PROGRAM MAIN
VAR
	// Invoker
	fbHMI_panel				: FB_ShowControlPanel;
	fbPendant_panel			: FB_ShowControlPanel;
	
	// Receiver
	fbFlyingHoist			: FB_FlyingHoist;
	refFlyingHoist			: REFERENCE TO FB_FlyingHoist := fbFlyingHoist;	
	fbFlameCannon			: FB_FlameCannon;
	refFlameCannon			: REFERENCE TO FB_FlameCannon := fbFlameCannon;	
	fbMovingHead			: FB_MovingHead;
	refMovingHead			: REFERENCE TO FB_MovingHead := fbMovingHead;	

	// Commands
	fbActorDownCommand			: FB_ActorDownCommand(refFlyingHoist);
	fbActorUpCommand			: FB_ActorUpCommand(refFlyingHoist);
	fbActorRotateCCWCommand		: FB_ActorRotateCCWCommand(refFlyingHoist);
	fbActorRotateCWCommand		: FB_ActorRotateCWCommand(refFlyingHoist);
	fbActorStopRotateCommand	: FB_ActorStopRotateCommand(refFlyingHoist);
	fbActorStopVerticalCommand	: FB_ActorStopVerticalCommand(refFlyingHoist);
	fbFireShowModeCommand		: FB_FireShowModeCommand(fbFlameCannon);
	fbFirePyroModeCommand		: FB_FireShowModeCommand(fbFlameCannon);
	fbFireOffCommand			: FB_FireOffCommand(fbFlameCannon);
	fbMovingHeadOnCommand		: FB_MovingHeadOnCommand(fbMovingHead);
	fbMovingHeadOffCommand		: FB_MovingHeadOffCommand(fbMovingHead);
	fbShowOnCommnad				: FB_ShowOnCommnad(fbActorUpCommand, fbActorRotateCWCommand, fbFireShowModeCommand);
	bInit						: BOOL;
	
	fHoistVertPos				: LREAL;
	fHoistRotPos				: LREAL;
END_VAR

IF (NOT bInit) THEN
	fbHMI_panel.SetCommand(1, fbActorDownCommand);
	fbHMI_panel.SetCommand(2, fbActorUpCommand);
	fbHMI_panel.SetCommand(3, fbActorRotateCCWCommand);
	fbHMI_panel.SetCommand(4, fbActorRotateCWCommand);
	fbHMI_panel.SetCommand(5, fbActorStopVerticalCommand);
	fbHMI_panel.SetCommand(6, fbActorStopRotateCommand);
	fbHMI_panel.SetCommand(7, fbFireShowModeCommand);
	fbHMI_panel.SetCommand(8, fbFirePyroModeCommand);
	fbHMI_panel.SetCommand(9, fbFireOffCommand);
	fbHMI_panel.SetCommand(10, fbMovingHeadOnCommand);
	fbHMI_panel.SetCommand(11, fbMovingHeadOffCommand);
	fbHMI_panel.SetCommand(12, fbShowOnCommnad);
	
	fbPendant_panel.SetCommand(1, fbActorDownCommand);
	fbPendant_panel.SetCommand(2, fbActorUpCommand);
	fbPendant_panel.SetCommand(3, fbActorRotateCCWCommand);
	fbPendant_panel.SetCommand(4, fbActorRotateCWCommand);
	fbPendant_panel.SetCommand(5, fbActorStopVerticalCommand);
	fbPendant_panel.SetCommand(6, fbActorStopRotateCommand);

	
	bInit := TRUE;
ELSE
	fbHMI_panel();	
	fbPendant_panel();
END_IF


(* Trigger fbPendant_panel.arrSwitch[1 - 4] for moves, and arrSwitch[5 - 6] for stops.
OR
Trigger fbHMI_panel.arrSwitch[1 - 4] for moves, and arrSwitch[5 - 6] for stops. *)

// Check the positions of the hoist
fHoistRotPos 	:= fbFlyingHoist.RotationalPosition;
fHoistVertPos 	:= fbFlyingHoist.VerticalPosition;

END_PROGRAM

(* stored: Version 1.1.0.1, ProductVersion 3.1.4022.18
   POU MAIN: Id {e55fe8ab-45d1-4feb-a2af-4eb48f72a41c}, SpecialFunc None *)
